FUNCTION_BLOCK "_teachPinPositionValues"
TITLE = {"version":"v1.1","author":"cyanezf","family":"core/control/util","status":"current","deprecatedBy": null,"dependencies" : []}
{ S7_Optimized_Access := 'TRUE' }
AUTHOR : cyanezf
FAMILY : 'core/control/util'
NAME : _teachPinPositionValues
VERSION : 1.1

   VAR_INPUT
      pin { ExternalWritable := 'False'} : Bool;   // IR: Pin sensor
      position { ExternalWritable := 'False'} : LReal;   // IR: Current position
      direction { ExternalWritable := 'False'} : Bool;   // IR: 0=Forward; 1=Backward
   END_VAR

   VAR_OUTPUT
      fwdPosEdgePosition { ExternalWritable := 'False'} : LReal;   // OR: Forward positive edge position
      fwdNegEdgePosition { ExternalWritable := 'False'} : LReal;   // OR: Forward negative edge position
      bwdPosEdgePosition { ExternalWritable := 'False'} : LReal;   // OR: Backward positive edge position
      bwdNegEdgePosition { ExternalWritable := 'False'} : LReal;   // OR: Backward negative edge position
   END_VAR

   VAR
      fp { ExternalAccessible := 'False'; ExternalVisible := 'False'; ExternalWritable := 'False'} : Bool;   // SX: Private static variables
   END_VAR

   VAR_TEMP
      pinFp : Bool;
      pinFn : Bool;
   END_VAR


BEGIN
(*--
# Documentation

## Log

| version | date | author | description |
|:-------:|:----:|:------:|:------------|
| v1.1 | 2026-06-17 | cyanezf | refactor: Change REAL with LREAL |
| v1.0 | 2024-02-15 | cyanezf | First version |

## Description

This function catches the position when `pin` sensor edges are detected in forward and backward direction.

--*)

	// Update edges
	#pinFp := #pin AND NOT #fp;
	#pinFn := NOT #pin AND #fp;
	#fp := #pin;

	IF #pinFp AND NOT #direction THEN
	  #fwdPosEdgePosition := #position;
	END_IF;

	IF #pinFp AND #direction THEN
	  #bwdPosEdgePosition := #position;
	END_IF;

	IF #pinFn AND NOT #direction THEN
	  #fwdNegEdgePosition := #position;
	END_IF;

	IF #pinFn AND #direction THEN
	  #bwdNegEdgePosition := #position;
	END_IF;

	// Savel RLO
	ENO := true;

END_FUNCTION_BLOCK

